PROGRAM BackgroundEL
VAR
	/// background communication with the EL6001 terminal 
	fbEL6001Ctrl: SerialLineControl;
	bEL6001CtrlError: BOOL;
	eEL6001CtrlErrorID: ComError_t;
	/// linked to the EL6001 in the TwinCAT System Manager 
	stIn_EL6001 AT %I*: EL6inData22B;
	/// linked to the EL6001 in the TwinCAT System Manager 
	stOut_EL6001 AT %Q*: EL6outData22B;
END_VAR

(*
The SerialLineControl function block is supposed to be called in every PLC cycle.
It communicates with the serial line hardware device and transmits or receives data.
The SerialLineControl can be called in the standard task (e.g.for PcCOM port usage) 
or in a separate fast task (e.g.for terminal usage) as well.
A fast separate task will be necessary at high baud rates or with KL6001 terminals 
which have a small process image (3 or 5 data bytes only)
*)

(* background communication with the EL6001 terminal *)
fbEL6001Ctrl(
	Mode:= SERIALLINEMODE_EL6_22B, 
	pComIn:= ADR(stIn_EL6001), 
	pComOut:= ADR(stOut_EL6001), 
	SizeComIn:= SIZEOF(stIn_EL6001), 
	Error=> , 
	ErrorID=> , 
	TxBuffer:= BuffTX, 
	RxBuffer:= BuffRX );
IF fbEL6001Ctrl.Error THEN
	bEL6001CtrlError := TRUE;
	eEL6001CtrlErrorID := fbEL6001Ctrl.ErrorID;
END_IF

END_PROGRAM

(* stored: Version 1.1.0.1, ProductVersion 3.1.0.26
   POU BackgroundEL: Id {abab1503-5149-4078-84ca-9b2293509a86} *)
